{attribute 'GeneratedUsingTerminal: EL2535-0000-0016'}
{attribute addProperty BoxType "EL2535-0000-0016"}
{attribute addProperty Id "Digital_input_1BOOL1Ready_to_enableBOOL1WarningBOOL1ErrorBOOL1TxPDO_ToggleBOOL1"}
{attribute addProperty CRC "3955946476"}
{attribute addProperty Size "5"}
TYPE Status_EBCAF3EC :
STRUCT
	{attribute addProperty Name "Digital_input_1"}
	Digital_input_1 : BOOL;
	{attribute addProperty Name "Ready_to_enable"}
	Ready_to_enable : BOOL;
	{attribute addProperty Name "Warning"}
	Warning : BOOL;
	{attribute addProperty Name "Error"}
	Error : BOOL;
	{attribute addProperty Name "TxPDO_Toggle"}
	TxPDO_Toggle : BOOL;
END_STRUCT
END_TYPE

(* stored: Version 1.2.0.0, ProductVersion 3.1.4024.9
   DUT Status_EBCAF3EC: Id {557f610d-1764-42a0-8084-147f171525b7} *)
